(* Logix 5000 project; controller SX_V040001_C001 vendor 1 type 14 code 77 rev 16.22; software revision 16.04; part 8 of 35 *)
(* tags used below, declared in another part *)
   ALL_KINDS : INT[90];
   ANA_OUTPUT_SIM : INT[8];
   CMD : INT[36];
   command_number : INT;
   DB_A_IO : INT[16];
   DIGI_OUTPUT_SIM : DINT[3];
   DIGI_OUTPUT_SIM_REVERSE : DINT[3];
   DRIVE : INT[32];
   DRIVE_INTERVAL : INT[8];
   EMPTYING : INT[18];
   G_AOutput : DINT[8];
   G_DInput : DINT[3];
   G_DOutput : DINT[3];
   loading : INT[19];
   m_on_off_line : BOOL;
   METERING : INT[44];
   PARAMETER : INT[501];
   pointer_bcc_in : DINT;
   pointer_bcc_out : DINT;
   REMOTE_DATA_IN : INT[510];
   REMOTE_DATA_OUT : INT[510];
   TEMP : INT[14];
   temp_bcc_in : DINT;
   temp_bcc_out : DINT;
(* MainProgram, continued *)

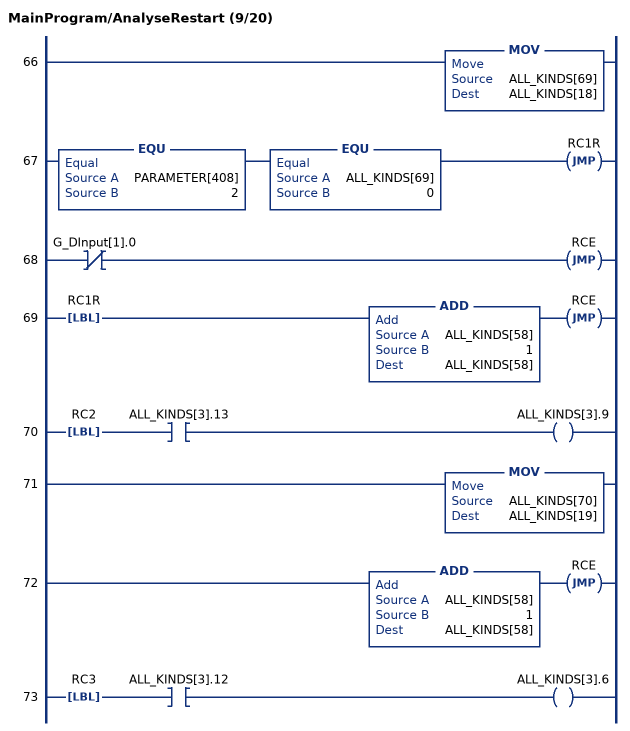
   [picture p166: MainProgram/AnalyseRestart rungs 66-73]
   66: MOV(ALL_KINDS[69],ALL_KINDS[18]);
   67: EQU(PARAMETER[408],2)EQU(ALL_KINDS[69],0)JMP(RC1R);
   68: XIO(G_DInput[1].0)JMP(RCE);
   69: LBL(RC1R)ADD(ALL_KINDS[58],1,ALL_KINDS[58])JMP(RCE);
   70: LBL(RC2)XIC(ALL_KINDS[3].13)OTE(ALL_KINDS[3].9);
   71: MOV(ALL_KINDS[70],ALL_KINDS[19]);
   72: ADD(ALL_KINDS[58],1,ALL_KINDS[58])JMP(RCE);
   73: LBL(RC3)XIC(ALL_KINDS[3].12)OTE(ALL_KINDS[3].6);
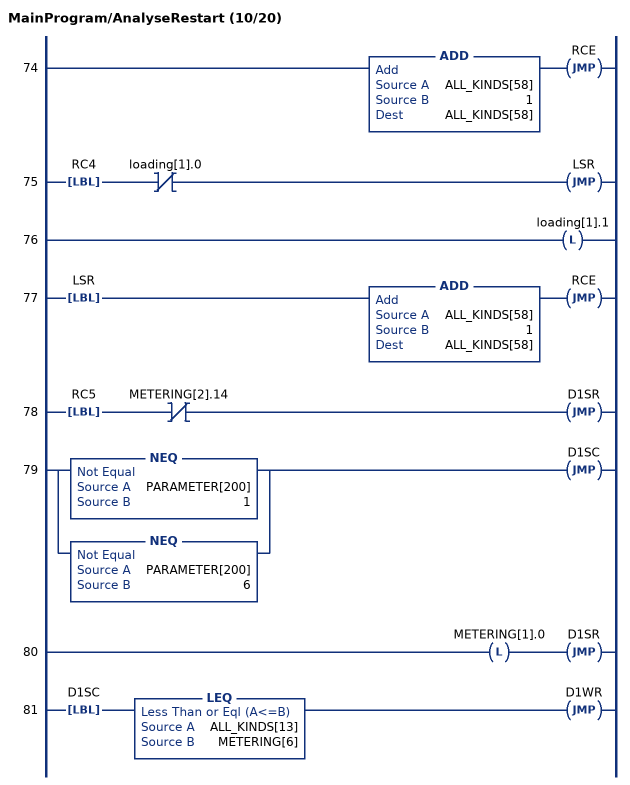
   74: ADD(ALL_KINDS[58],1,ALL_KINDS[58])JMP(RCE);
   75: LBL(RC4)XIO(loading[1].0)JMP(LSR);
   76: OTL(loading[1].1);
   77: LBL(LSR)ADD(ALL_KINDS[58],1,ALL_KINDS[58])JMP(RCE);
   78: LBL(RC5)XIO(METERING[2].14)JMP(D1SR);
   79: [NEQ(PARAMETER[200],1) ,NEQ(PARAMETER[200],6) ]JMP(D1SC);
   80: OTL(METERING[1].0)JMP(D1SR);
   81: LBL(D1SC)LEQ(ALL_KINDS[13],METERING[6])JMP(D1WR);
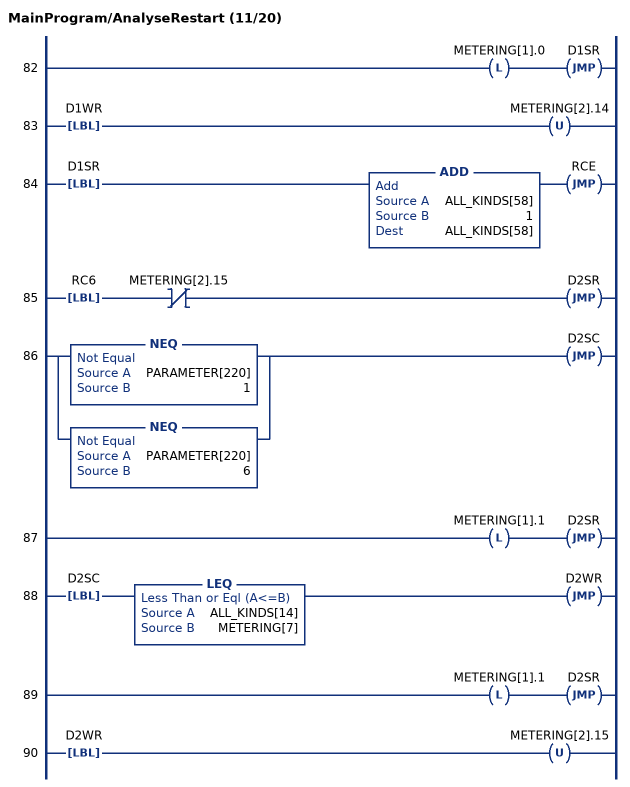
   82: OTL(METERING[1].0)JMP(D1SR);
   83: LBL(D1WR)OTU(METERING[2].14);
   84: LBL(D1SR)ADD(ALL_KINDS[58],1,ALL_KINDS[58])JMP(RCE);
   85: LBL(RC6)XIO(METERING[2].15)JMP(D2SR);
   86: [NEQ(PARAMETER[220],1) ,NEQ(PARAMETER[220],6) ]JMP(D2SC);
   87: OTL(METERING[1].1)JMP(D2SR);
   88: LBL(D2SC)LEQ(ALL_KINDS[14],METERING[7])JMP(D2WR);
   89: OTL(METERING[1].1)JMP(D2SR);
   90: LBL(D2WR)OTU(METERING[2].15);
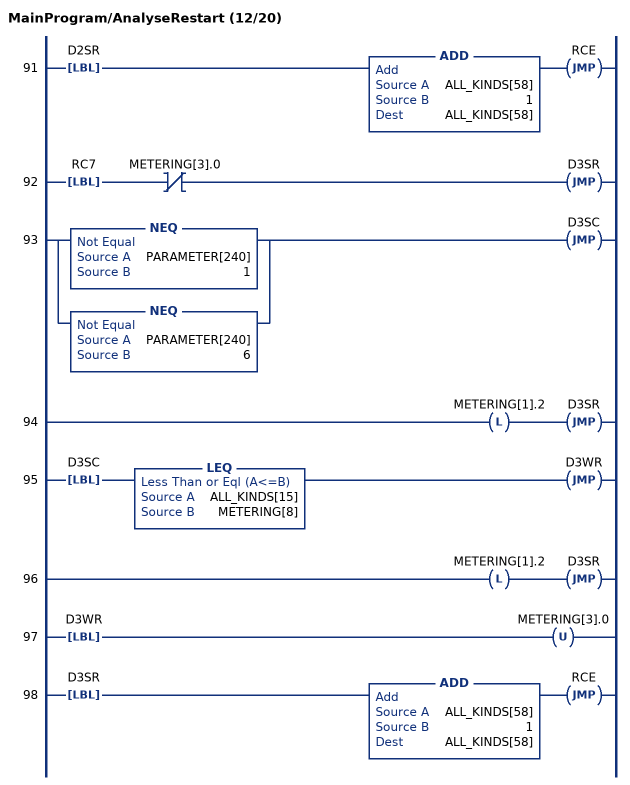
   91: LBL(D2SR)ADD(ALL_KINDS[58],1,ALL_KINDS[58])JMP(RCE);
   92: LBL(RC7)XIO(METERING[3].0)JMP(D3SR);
   93: [NEQ(PARAMETER[240],1) ,NEQ(PARAMETER[240],6) ]JMP(D3SC);
   94: OTL(METERING[1].2)JMP(D3SR);
   95: LBL(D3SC)LEQ(ALL_KINDS[15],METERING[8])JMP(D3WR);
   96: OTL(METERING[1].2)JMP(D3SR);
   97: LBL(D3WR)OTU(METERING[3].0);
   98: LBL(D3SR)ADD(ALL_KINDS[58],1,ALL_KINDS[58])JMP(RCE);
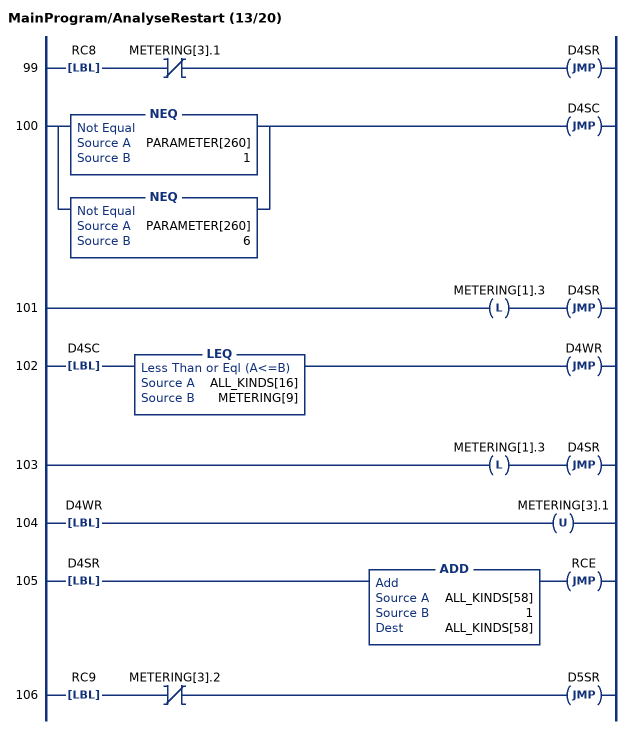
   99: LBL(RC8)XIO(METERING[3].1)JMP(D4SR);
   100: [NEQ(PARAMETER[260],1) ,NEQ(PARAMETER[260],6) ]JMP(D4SC);
   101: OTL(METERING[1].3)JMP(D4SR);
   102: LBL(D4SC)LEQ(ALL_KINDS[16],METERING[9])JMP(D4WR);
   103: OTL(METERING[1].3)JMP(D4SR);
   104: LBL(D4WR)OTU(METERING[3].1);
   105: LBL(D4SR)ADD(ALL_KINDS[58],1,ALL_KINDS[58])JMP(RCE);
   106: LBL(RC9)XIO(METERING[3].2)JMP(D5SR);
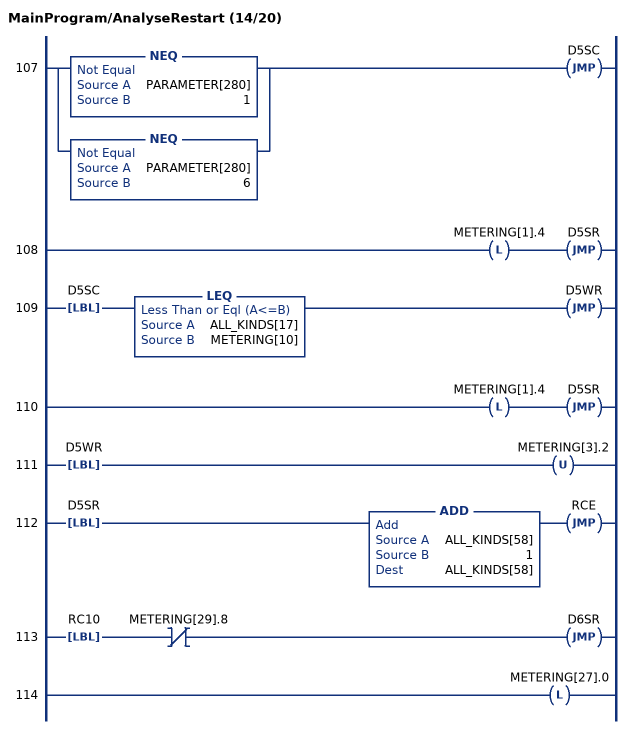
   107: [NEQ(PARAMETER[280],1) ,NEQ(PARAMETER[280],6) ]JMP(D5SC);
   108: OTL(METERING[1].4)JMP(D5SR);
   109: LBL(D5SC)LEQ(ALL_KINDS[17],METERING[10])JMP(D5WR);
   110: OTL(METERING[1].4)JMP(D5SR);
   111: LBL(D5WR)OTU(METERING[3].2);
   112: LBL(D5SR)ADD(ALL_KINDS[58],1,ALL_KINDS[58])JMP(RCE);
   113: LBL(RC10)XIO(METERING[29].8)JMP(D6SR);
   114: OTL(METERING[27].0);
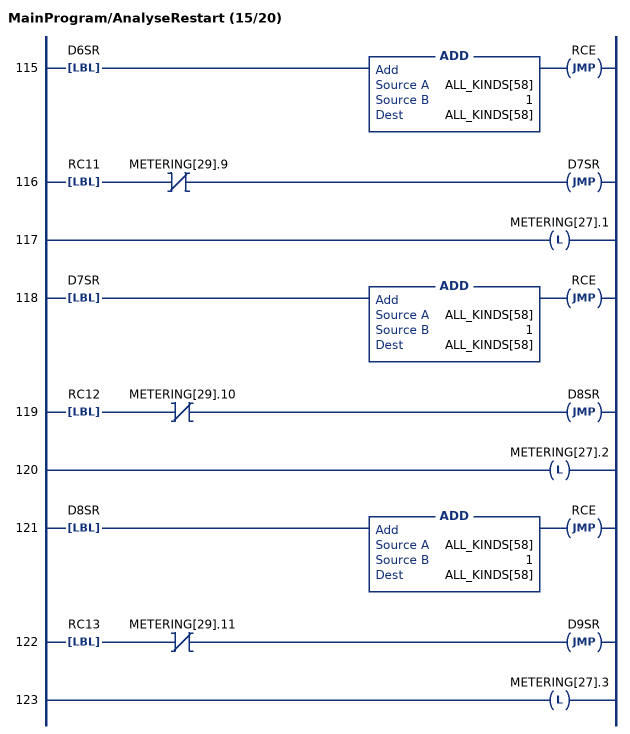
   115: LBL(D6SR)ADD(ALL_KINDS[58],1,ALL_KINDS[58])JMP(RCE);
   116: LBL(RC11)XIO(METERING[29].9)JMP(D7SR);
   117: OTL(METERING[27].1);
   118: LBL(D7SR)ADD(ALL_KINDS[58],1,ALL_KINDS[58])JMP(RCE);
   119: LBL(RC12)XIO(METERING[29].10)JMP(D8SR);
   120: OTL(METERING[27].2);
   121: LBL(D8SR)ADD(ALL_KINDS[58],1,ALL_KINDS[58])JMP(RCE);
   122: LBL(RC13)XIO(METERING[29].11)JMP(D9SR);
   123: OTL(METERING[27].3);
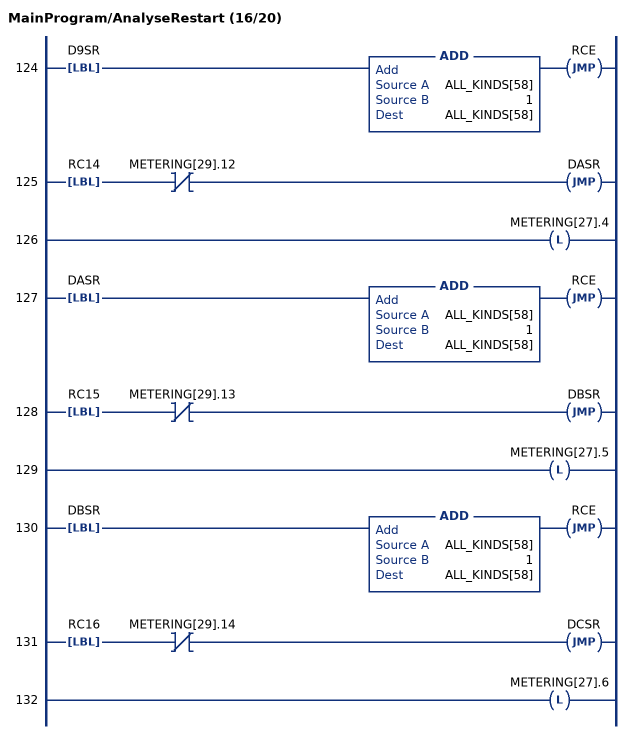
   124: LBL(D9SR)ADD(ALL_KINDS[58],1,ALL_KINDS[58])JMP(RCE);
   125: LBL(RC14)XIO(METERING[29].12)JMP(DASR);
   126: OTL(METERING[27].4);
   127: LBL(DASR)ADD(ALL_KINDS[58],1,ALL_KINDS[58])JMP(RCE);
   128: LBL(RC15)XIO(METERING[29].13)JMP(DBSR);
   129: OTL(METERING[27].5);
   130: LBL(DBSR)ADD(ALL_KINDS[58],1,ALL_KINDS[58])JMP(RCE);
   131: LBL(RC16)XIO(METERING[29].14)JMP(DCSR);
   132: OTL(METERING[27].6);
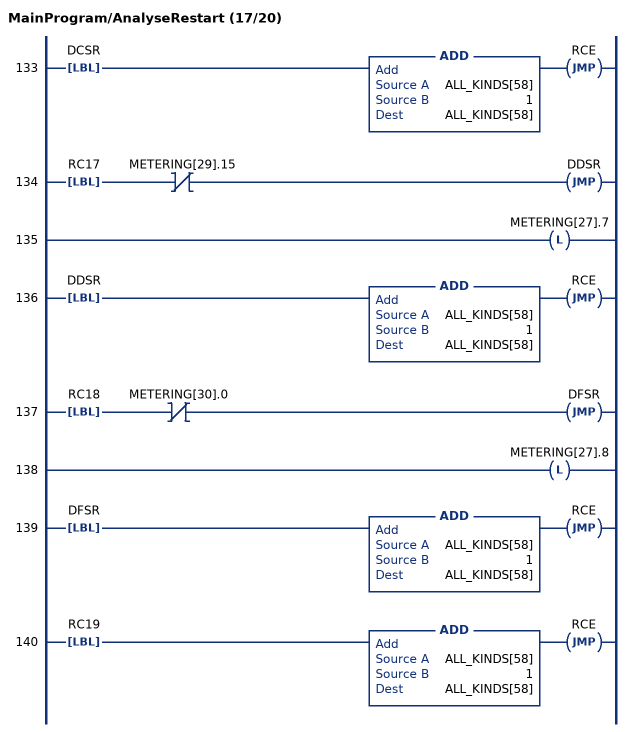
   133: LBL(DCSR)ADD(ALL_KINDS[58],1,ALL_KINDS[58])JMP(RCE);
   134: LBL(RC17)XIO(METERING[29].15)JMP(DDSR);
   135: OTL(METERING[27].7);
   136: LBL(DDSR)ADD(ALL_KINDS[58],1,ALL_KINDS[58])JMP(RCE);
   137: LBL(RC18)XIO(METERING[30].0)JMP(DFSR);
   138: OTL(METERING[27].8);
   139: LBL(DFSR)ADD(ALL_KINDS[58],1,ALL_KINDS[58])JMP(RCE);
   140: LBL(RC19)ADD(ALL_KINDS[58],1,ALL_KINDS[58])JMP(RCE);
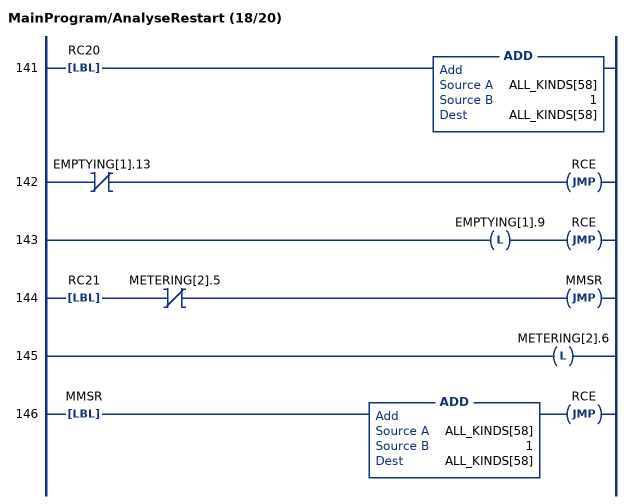
   141: LBL(RC20)ADD(ALL_KINDS[58],1,ALL_KINDS[58]);
   142: XIO(EMPTYING[1].13)JMP(RCE);
   143: OTL(EMPTYING[1].9)JMP(RCE);
   144: LBL(RC21)XIO(METERING[2].5)JMP(MMSR);
   145: OTL(METERING[2].6);
   146: LBL(MMSR)ADD(ALL_KINDS[58],1,ALL_KINDS[58])JMP(RCE);
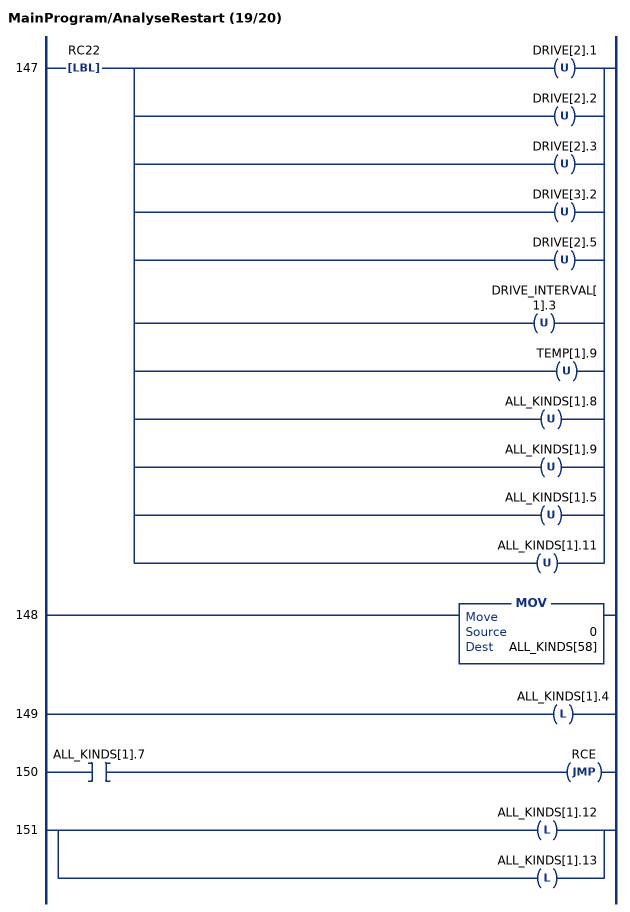
   147: LBL(RC22)[OTU(DRIVE[2].1) ,OTU(DRIVE[2].2) ,OTU(DRIVE[2].3) ,OTU(DRIVE[3].2) ,OTU(DRIVE[2].5) ,OTU(DRIVE_INTERVAL[1].3) ,OTU(TEMP[1].9) ,OTU(ALL_KINDS[1].8) ,OTU(ALL_KINDS[1].9) ,OTU(ALL_KINDS[1].5) ,OTU(ALL_KINDS[1].11) ];
   148: MOV(0,ALL_KINDS[58]);
   149: OTL(ALL_KINDS[1].4);
   150: XIC(ALL_KINDS[1].7)JMP(RCE);
   151: [OTL(ALL_KINDS[1].12) ,OTL(ALL_KINDS[1].13) ];
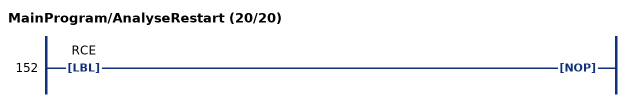
   152: LBL(RCE)NOP();
END_ROUTINE

ROUTINE CalcBCC_IN   (* ladder *)
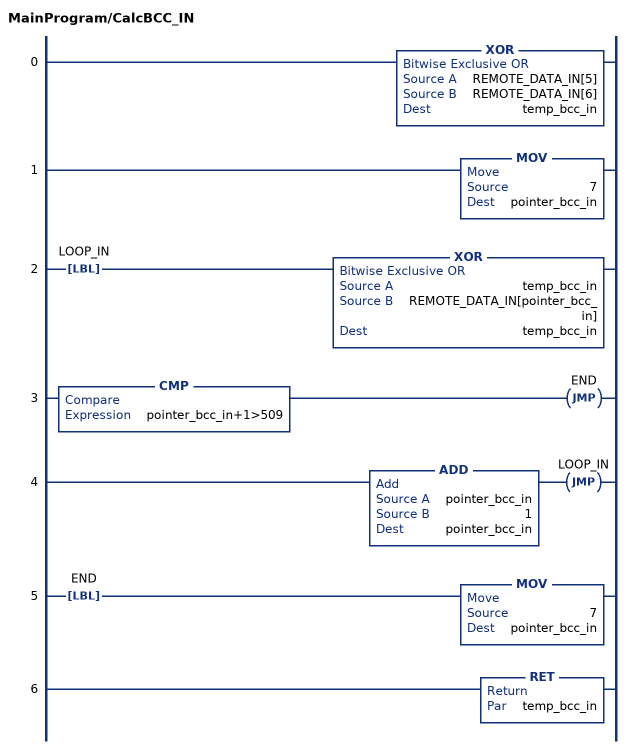
   0: XOR(REMOTE_DATA_IN[5],REMOTE_DATA_IN[6],temp_bcc_in);
   1: MOV(7,pointer_bcc_in);
   2: LBL(LOOP_IN)XOR(temp_bcc_in,REMOTE_DATA_IN[pointer_bcc_in],temp_bcc_in);
   3: CMP(pointer_bcc_in+1>509)JMP(END);
   4: ADD(pointer_bcc_in,1,pointer_bcc_in)JMP(LOOP_IN);
   5: LBL(END)MOV(7,pointer_bcc_in);
   6: RET(temp_bcc_in);
END_ROUTINE

ROUTINE CalcBCC_OUT   (* ladder *)
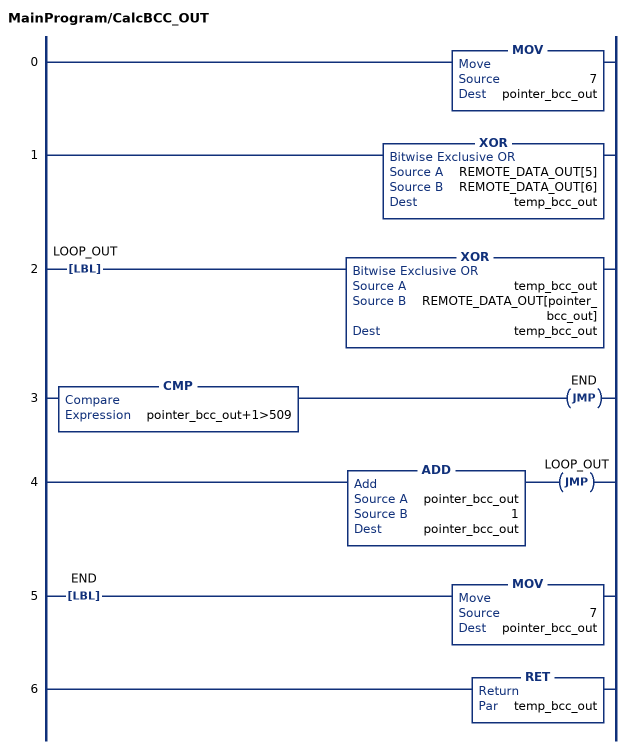
   0: MOV(7,pointer_bcc_out);
   1: XOR(REMOTE_DATA_OUT[5],REMOTE_DATA_OUT[6],temp_bcc_out);
   2: LBL(LOOP_OUT)XOR(temp_bcc_out,REMOTE_DATA_OUT[pointer_bcc_out],temp_bcc_out);
   3: CMP(pointer_bcc_out+1>509)JMP(END);
   4: ADD(pointer_bcc_out,1,pointer_bcc_out)JMP(LOOP_OUT);
   5: LBL(END)MOV(7,pointer_bcc_out);
   6: RET(temp_bcc_out);
END_ROUTINE

ROUTINE ComDeco_1   (* ladder *)
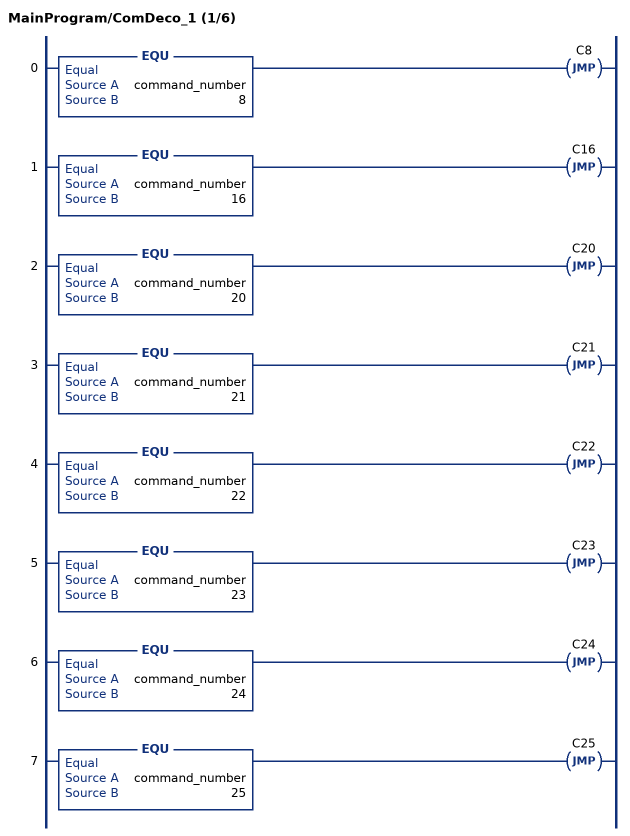
   0: EQU(command_number,8)JMP(C8);
   1: EQU(command_number,16)JMP(C16);
   2: EQU(command_number,20)JMP(C20);
   3: EQU(command_number,21)JMP(C21);
   4: EQU(command_number,22)JMP(C22);
   5: EQU(command_number,23)JMP(C23);
   6: EQU(command_number,24)JMP(C24);
   7: EQU(command_number,25)JMP(C25);
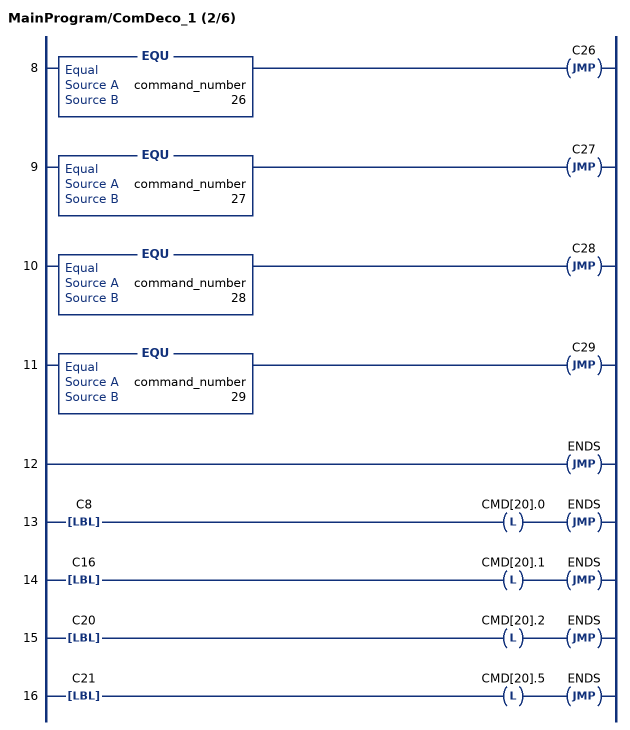
   8: EQU(command_number,26)JMP(C26);
   9: EQU(command_number,27)JMP(C27);
   10: EQU(command_number,28)JMP(C28);
   11: EQU(command_number,29)JMP(C29);
   12: JMP(ENDS);
   13: LBL(C8)OTL(CMD[20].0)JMP(ENDS);
   14: LBL(C16)OTL(CMD[20].1)JMP(ENDS);
   15: LBL(C20)OTL(CMD[20].2)JMP(ENDS);
   16: LBL(C21)OTL(CMD[20].5)JMP(ENDS);
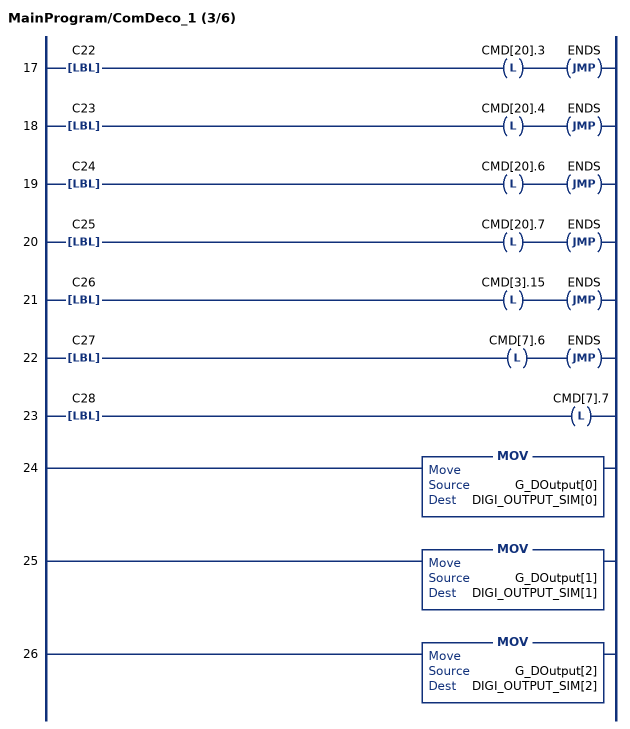
   17: LBL(C22)OTL(CMD[20].3)JMP(ENDS);
   18: LBL(C23)OTL(CMD[20].4)JMP(ENDS);
   19: LBL(C24)OTL(CMD[20].6)JMP(ENDS);
   20: LBL(C25)OTL(CMD[20].7)JMP(ENDS);
   21: LBL(C26)OTL(CMD[3].15)JMP(ENDS);
   22: LBL(C27)OTL(CMD[7].6)JMP(ENDS);
   23: LBL(C28)OTL(CMD[7].7);
   24: MOV(G_DOutput[0],DIGI_OUTPUT_SIM[0]);
   25: MOV(G_DOutput[1],DIGI_OUTPUT_SIM[1]);
   26: MOV(G_DOutput[2],DIGI_OUTPUT_SIM[2]);
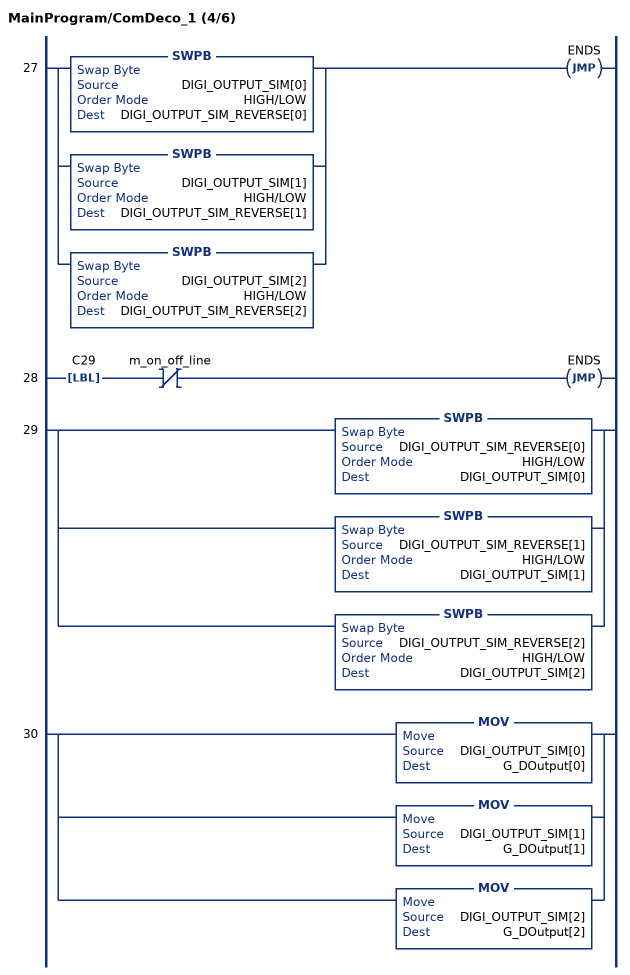
   27: [SWPB(DIGI_OUTPUT_SIM[0],HIGH/LOW,DIGI_OUTPUT_SIM_REVERSE[0]) ,SWPB(DIGI_OUTPUT_SIM[1],HIGH/LOW,DIGI_OUTPUT_SIM_REVERSE[1]) ,SWPB(DIGI_OUTPUT_SIM[2],HIGH/LOW,DIGI_OUTPUT_SIM_REVERSE[2]) ]JMP(ENDS);
   28: LBL(C29)XIO(m_on_off_line)JMP(ENDS);
   29: [SWPB(DIGI_OUTPUT_SIM_REVERSE[0],HIGH/LOW,DIGI_OUTPUT_SIM[0]) ,SWPB(DIGI_OUTPUT_SIM_REVERSE[1],HIGH/LOW,DIGI_OUTPUT_SIM[1]) ,SWPB(DIGI_OUTPUT_SIM_REVERSE[2],HIGH/LOW,DIGI_OUTPUT_SIM[2]) ];
   30: [MOV(DIGI_OUTPUT_SIM[0],G_DOutput[0]) ,MOV(DIGI_OUTPUT_SIM[1],G_DOutput[1]) ,MOV(DIGI_OUTPUT_SIM[2],G_DOutput[2]) ];
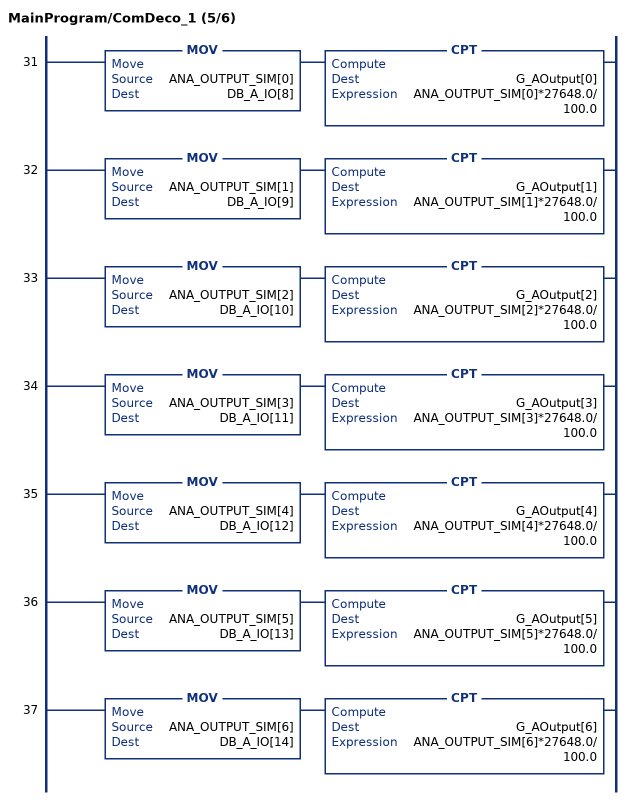
   31: MOV(ANA_OUTPUT_SIM[0],DB_A_IO[8])CPT(G_AOutput[0],ANA_OUTPUT_SIM[0]*27648.0/100.0);
   32: MOV(ANA_OUTPUT_SIM[1],DB_A_IO[9])CPT(G_AOutput[1],ANA_OUTPUT_SIM[1]*27648.0/100.0);
   33: MOV(ANA_OUTPUT_SIM[2],DB_A_IO[10])CPT(G_AOutput[2],ANA_OUTPUT_SIM[2]*27648.0/100.0);
   34: MOV(ANA_OUTPUT_SIM[3],DB_A_IO[11])CPT(G_AOutput[3],ANA_OUTPUT_SIM[3]*27648.0/100.0);
   35: MOV(ANA_OUTPUT_SIM[4],DB_A_IO[12])CPT(G_AOutput[4],ANA_OUTPUT_SIM[4]*27648.0/100.0);
   36: MOV(ANA_OUTPUT_SIM[5],DB_A_IO[13])CPT(G_AOutput[5],ANA_OUTPUT_SIM[5]*27648.0/100.0);
   37: MOV(ANA_OUTPUT_SIM[6],DB_A_IO[14])CPT(G_AOutput[6],ANA_OUTPUT_SIM[6]*27648.0/100.0);
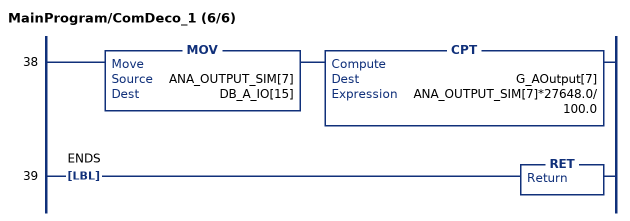
   38: MOV(ANA_OUTPUT_SIM[7],DB_A_IO[15])CPT(G_AOutput[7],ANA_OUTPUT_SIM[7]*27648.0/100.0);
   39: LBL(ENDS)RET();
END_ROUTINE
